FUNCTION_BLOCK FB_Car
VAR_INPUT
END_VAR
VAR
	sCarName : STRING(300);
	fRunning : BOOL;
END_VAR

METHOD SetCarName : REFERENCE TO FB_Car
VAR_INPUT
	sCarName : STRING(300);
END_VAR
THIS^.sCarName := sCarName;
SetCarName REF= THIS^;
END_METHOD

METHOD Start : BOOL
VAR_INPUT
END_VAR
fRunning := TRUE;
END_METHOD

END_FUNCTION_BLOCK

(* stored: Version 1.1.0.1, ProductVersion 3.1.4024.16
   POU FB_Car: Id {5fe7ec5a-d238-4042-ad4a-826fc3508585}, SpecialFunc None
   Method SetCarName: Id {6261db08-61dc-413c-9bbc-d64417642136}
   Method Start: Id {ee051c42-472a-4eec-9947-e2706b965e6f} *)
